TYPE UDT_RackFeedMessage_RD :
STRUCT
tail : BOOL; // 尾料模式，缺料时不提示
timeoutAlarm : BOOL; // 放料超时报警
breakAlarm : BOOL; // 纸带断裂报警
scatterAlarm : BOOL; // 散料报警

END_STRUCT
END_TYPE

(* stored: Version 1.1.0.1, ProductVersion 3.1.4024.12
   DUT UDT_RackFeedMessage_RD: Id {357d8b82-4fd0-4f40-ab56-a5e14b4315ed} *)
